KUKA KRL program: CadMatchExample.src, CadMatchExample.dat

--- CadMatchExample.src ---
&ACCESS RVO
&REL 1
&PARAM DISKPATH = KRC:\R1\Program

DEF CadMatchExample()
   ;------------------------------------------------------------------------
   ; CADMatch Example Program for Roboception rc_visard/rc_cube
   ;
   ; This program demonstrates CAD-based object detection and pick-and-place
   ; operations using Roboception's CADMatch module. The program:
   ; 1. Configures detection parameters for the specified template
   ; 2. Performs object detection with retry mechanism
   ; 3. Executes pick-and-place operations for detected objects
   ; 4. Continues until no more objects are found or program is interrupted
   ;
   ; IMPORTANT SETUP INSTRUCTIONS:
   ; 1. The service names MUST match exactly with your EKI XML configuration files
   ; 2. Modify only the parameters in this section before running the program
   ; 3. Teach the STARTPOSE and PLACEPOSE positions in the .dat file
   ; 4. Define the GripperClose() and GripperOpen() functions for your specific gripper
   ;
   ; HOW THE PROGRAM WORKS:
   ; - The program calls the CADMatch detection service which returns an array of possible grasps
   ; - Currently, only the first grasp (index 1) is used for the pick-and-place sequence
   ; - The program reads the gripper_id associated with the first grasp.
   ; - Based on the gripper_id, a target opening value is determined.
   ; - If detection fails, the program will retry up to MAX_DETECTION_RETRIES times
   ; - After successful detection, the robot will:
   ;   a) Move to a pre-grasp position above the detected object
   ;   b) Move down to grasp the object
   ;   c) Pick up the object and move to the pre-place position
   ;   d) Place the object at the taught PLACEPOSE
   ;   e) Return to the start position and repeat the cycle
   ;
   ; To use multiple detected objects, you would need to modify the code to
   ; iterate through the DETECTEDGRASPS array (indices 1 to NUMDETECTEDGRASPS)
   ;------------------------------------------------------------------------
   DECL INT MAX_DETECTION_RETRIES
   DECL INT RETRY_COUNT
   DECL REAL targetOpening      ; Calculated target opening for the gripper
   DECL REAL defaultOpening     ; Default opening value
   DECL CHAR tempMsg[120]       ; Temporary buffer for constructing messages
   DECL STATE_T State           ; State variable for SWRITE
   DECL INT Offset              ; Offset variable for SWRITE
   DECL E6POS selectedPlacePose ; Stores the selected place pose

   ; Service name - same as the EKI service name
   ; TODO: Change this to the correct service name - could be "sensor_a_pipeline_1_rc_cadmatch-detect_object"
   serviceNameDetect[] = "rc_cadmatch-detect_object"
   serviceNameStart[] = "rc_cadmatch-start"
   serviceNameStop[] = "rc_cadmatch-stop"

   ; Detection configuration parameters
   TEMPLATE_ID[] = "Template_Name"         ; CAD template to match
   POSE_FRAME[] = "external"               ; Reference frame for poses
   LOAD_CARRIER_ID[] = " "                 ; Load carrier ID (Whitespace " " = none)
   ROI_ID[] = " "                          ; Region of interest ID

   ; Collision checking parameters - deactivate all to disable collision checking
   GRIPPER_ID[] = " "                      ; Gripper ID for collision checking
   ; Pre-grasp offset for collision checking (in meters) - negtive vlaues normally desired
   PRE_GRASP_OFFSET_X = 0.0                 ; X offset - set to 0 to disable
   PRE_GRASP_OFFSET_Y = 0.0                 ; Y offset - set to 0 to disable
   PRE_GRASP_OFFSET_Z = -0.3                ; Z offset - set to 0 to disable

   ; Motion parameters (in millimeters)
   MOT_PRE_GRASP_Z_OFFSET = -300        ; Vertical offset for pre-grasp position
   MOT_PRE_PLACE_Z_OFFSET = -300        ; Vertical offset for pre-place position

   ; Detection retry configuration
   MAX_DETECTION_RETRIES = 3        ; Maximum number of detection attempts

   ; Gripper configuration
   defaultOpening = 100.0           ; Set your default gripper opening here

   ; Initialize robot and set up interrupts
   ;FOLD INI
      ;FOLD BASISTECH INI
         GLOBAL INTERRUPT DECL 3 WHEN $STOPMESS==TRUE DO IR_STOPM()
         INTERRUPT ON 3
         BAS(#INITMOV,0)
      ;ENDFOLD (BASISTECH INI)
   ;ENDFOLD (INI)

   ; Initialize message received interrupt for EKI communication
   INTERRUPT DECL 89 WHEN $FLAG[998] DO RC_NOTIFYRECEIVED(1, 998)
   INTERRUPT ON 89

   ; Move robot to home position and open gripper
   GripperOpen(defaultOpening)
   MoveToStartPosition()

   ; Initialize CADMatch module and open connection to rc_cube
   RC_START(serviceNameStart[])
   $FLAG[1] = FALSE
   RC_SETMSG("Start")

   RC_INIT(serviceNameDetect[])

   ; Main detection and pick-and-place loop
   LOOP
      ; Reset vision results
      ResetDetectedGrasps()
      RECEIVED_GRIPPER_ID[] = "none" ; Reset received ID for this cycle
      RECEIVED_GRASP_ID[] = "none"   ; Reset received grasp ID for this cycle
      targetOpening = defaultOpening   ; Reset target opening to default

      ; Attempt detection with retries
      FOR RETRY_COUNT = 1 TO MAX_DETECTION_RETRIES
         ; Pass all parameters to PerformDetection
         PerformDetection(serviceNameDetect[], TEMPLATE_ID[], POSE_FRAME[], LOAD_CARRIER_ID[], ROI_ID[], GRIPPER_ID[], PRE_GRASP_OFFSET_X, PRE_GRASP_OFFSET_Y, PRE_GRASP_OFFSET_Z)

         IF DetectionSuccessful() THEN
            RC_SETMSG("Detection successful")
            EXIT
         ENDIF

         IF RETRY_COUNT < MAX_DETECTION_RETRIES THEN
            ; Display the specific error message from RETURNCODE instead of generic one
            Offset = 0 ; Reset SWRITE offset
            SWRITE(tempMsg[], State, Offset, "Detection failed (Attempt %d/%d): %s Retrying...", RETRY_COUNT, MAX_DETECTION_RETRIES, RETURNCODE.MSG[])
            RC_SETMSG(tempMsg[])
            WAIT SEC 1.0  ; Brief delay between retries
         ENDIF
      ENDFOR

      IF DetectionSuccessful() THEN
         ; --- Gripper ID Logic ---
         ; Print the received gripper ID
         Offset = 0 ; Reset offset for SWRITE
         SWRITE(tempMsg[], State, Offset, "Received Gripper ID: %s", RECEIVED_GRIPPER_ID[])
         RC_SETMSG(tempMsg[])

         ; Print the received grasp ID
         Offset = 0 ; Reset offset for SWRITE
         SWRITE(tempMsg[], State, Offset, "Received Grasp ID: %s", RECEIVED_GRASP_ID[])
         RC_SETMSG(tempMsg[])

         ; Determine target opening based on ID
         IF STRCOMP(RECEIVED_GRIPPER_ID[], "gripper_a", #NOT_CASE_SENS) THEN
            targetOpening = 100.0
            RC_SETMSG("Gripper A identified, setting opening to 100.0")
         ELSE
            IF STRCOMP(RECEIVED_GRIPPER_ID[], "gripper_b", #NOT_CASE_SENS) THEN
               targetOpening = 50.0
               RC_SETMSG("Gripper B identified, setting opening to 50.0")
            ELSE
               ; Handle unknown or default case ("none" or other IDs)
               targetOpening = defaultOpening ; Use default opening
               RC_SETMSG("Unknown or default gripper ID, using default opening.")
            ENDIF
         ENDIF
         ; --- End Gripper ID Logic ---

         ; --- Place Pose Selection Logic based on Grasp ID ---

         IF STRCOMP(RECEIVED_GRASP_ID[], "grasp_1", #NOT_CASE_SENS) THEN
            selectedPlacePose = PLACEPOSE1 ; Assumes PLACEPOSE1 is defined in .dat
            RC_SETMSG("Grasp ID grasp_1 detected, using PLACEPOSE1.")
         ELSE
            IF STRCOMP(RECEIVED_GRASP_ID[], "grasp_2", #NOT_CASE_SENS) THEN
               selectedPlacePose = PLACEPOSE2 ; Assumes PLACEPOSE2 is defined in .dat
               RC_SETMSG("Grasp ID grasp_2 detected, using PLACEPOSE2.")
            ELSE
               selectedPlacePose = PLACEPOSE ; Use original PLACEPOSE as default
               RC_SETMSG("Unknown or default grasp ID, using default PLACEPOSE.")
            ENDIF
         ENDIF
         ; --- End Place Pose Selection Logic ---

         ExecutePickAndPlace(DETECTEDGRASPS[1], selectedPlacePose, MOT_PRE_GRASP_Z_OFFSET, MOT_PRE_PLACE_Z_OFFSET, targetOpening)
      ELSE
         HandleDetectionFailure()
         EXIT  ; Exit main loop if detection fails after all retries
      ENDIF
   ENDLOOP

   ; Clean up and stop the service
   RC_STOP(serviceNameStop[])
END

DEF ExecutePickAndPlace(GRASPPOSE:IN, PLACEPOSE:IN, MOT_PRE_GRASP_Z_OFFSET:IN, MOT_PRE_PLACE_Z_OFFSET:IN, targetOpening:IN)
   ; Executes a complete pick-and-place operation
   ;
   ; @param GRASPPOSE: Target pose for grasping the object
   ; @param PLACEPOSE: Target pose for placing the object
   ; @param MOT_PRE_GRASP_Z_OFFSET: Vertical offset (mm) for pre-grasp approach position
   ; @param MOT_PRE_PLACE_Z_OFFSET: Vertical offset (mm) for pre-place approach position
   ; @param targetOpening: The calculated opening value for the gripper

   DECL FRAME GRASPPOSE
   DECL E6POS PLACEPOSE
   DECL REAL MOT_PRE_GRASP_Z_OFFSET, MOT_PRE_PLACE_Z_OFFSET
   DECL REAL targetOpening

   ; Internal pose calculations
   DECL FRAME PREGRASPPOSE, PREPLACEPOSE
   DECL FRAME F_OFFSET

   ; Calculate pre-grasp pose using frame offset
   F_OFFSET = $NULLFRAME
   F_OFFSET.Z = MOT_PRE_GRASP_Z_OFFSET
   PREGRASPPOSE = GRASPPOSE:F_OFFSET

   ; Calculate pre-place pose
   PREPLACEPOSE = PLACEPOSE
   PREPLACEPOSE.z = PLACEPOSE.z + MOT_PRE_PLACE_Z_OFFSET

   ; Move to pre-grasp position
   SPTP PREGRASPPOSE WITH $VEL_AXIS[1] = SVEL_JOINT(rptpVelocityStd), $TOOL = STOOL2(fDatDefault), $BASE = SBASE(fDatDefault.BASE_NO), $IPO_MODE = SIPO_MODE(fDatDefault.IPO_FRAME), $LOAD = SLOAD(fDatDefault.TOOL_NO), $ACC_AXIS[1] = SACC_JOINT(pDatDefault), $APO = SAPO_PTP(pDatDefault), $GEAR_JERK[1] = SGEAR_JERK(pDatDefault)

   ; Open gripper before final approach (optional, might be already open)
   ; GripperOpen(targetOpening) ; Consider if needed here or rely on initial open

   ; Move to grasp position
   SLIN GRASPPOSE WITH $VEL = SVEL_CP(rlinVelocitySlow, , lDatDefault), $TOOL = STOOL2(fDatDefault), $BASE = SBASE(fDatDefault.BASE_NO)

   ; Activate gripper
   GripperClose()

   ; Add a small wait if needed for gripper to physically close
   WAIT SEC 0.5 ; Adjust timing as needed

   ; Optional: Add grasp check logic here if available for your gripper

   ; Move back to pre-grasp position
   SLIN PREGRASPPOSE WITH $VEL = SVEL_CP(rlinVelocityStd, , lDatDefault), $TOOL = STOOL2(fDatDefault), $BASE = SBASE(fDatDefault.BASE_NO)

   ; Move to pre-place position
   SPTP PREPLACEPOSE WITH $VEL_AXIS[1] = SVEL_JOINT(rptpVelocityStd), $TOOL = STOOL2(fDatDefault), $BASE = SBASE(fDatDefault.BASE_NO), $IPO_MODE = SIPO_MODE(fDatDefault.IPO_FRAME), $LOAD = SLOAD(fDatDefault.TOOL_NO), $ACC_AXIS[1] = SACC_JOINT(pDatDefault), $APO = SAPO_PTP(pDatDefault), $GEAR_JERK[1] = SGEAR_JERK(pDatDefault)

   ; Move to place position (user-taught position)
   ;FOLD LIN PLACEPOSE Vel=0.2 m/s CPDAT1 Tool[0]:Magnet Base[0] ;%{PE}
      ;FOLD Parameters ;%{h}
         ;Params IlfProvider=kukaroboter.basistech.inlineforms.movement.old; Kuka.IsGlobalPoint=False; Kuka.PointName=P4; Kuka.BlendingEnabled=False; Kuka.MoveDataName=CPDAT1; Kuka.VelocityPath=0.2; Kuka.CurrentCDSetIndex=0; Kuka.MovementParameterFieldEnabled=True; IlfCommand=LIN
      ;ENDFOLD
      $BWDSTART = FALSE
      LDAT_ACT = lDatDefault
      FDAT_ACT = fDatDefault
      BAS(#CP_PARAMS, 0.2)
      SET_CD_PARAMS(0)
      LIN PLACEPOSE
   ;ENDFOLD

   ; Release object
   GripperOpen(targetOpening)

   ; Add a small wait if needed for gripper to physically open
   WAIT SEC 0.5 ; Adjust timing as needed

   ; Move back to pre-place position
   SLIN PREPLACEPOSE WITH $VEL = SVEL_CP(rlinVelocityStd, , lDatDefault), $TOOL = STOOL2(fDatDefault), $BASE = SBASE(fDatDefault.BASE_NO)

   ; Return to home position
   MoveToStartPosition()
END

; ---- Helper Functions ----
DEF MoveToStartPosition()
   ;FOLD SPTP STARTPOSE Vel=100 % DEFAULT
      SPTP STARTPOSE WITH $VEL_AXIS[1]= SVEL_JOINT(100), $TOOL= STOOL2(fDatDefault), $BASE= SBASE(fDatDefault.BASE_NO), $IPO_MODE= SIPO_MODE(fDatDefault.IPO_FRAME), $LOAD= SLOAD(fDatDefault.TOOL_NO), $ACC_AXIS[1]= SACC_JOINT(PDEFAULT), $GEAR_JERK[1]= SGEAR_JERK(PDEFAULT)
   ;ENDFOLD
END

DEF GripperClose()
   ; Implement gripper closing logic here
   RC_SETMSG("Gripper closing")
   ; Example: SetOutput(GripperCloseSignal, TRUE)
   ; Example: SetOutput(GripperOpenSignal, FALSE)
   WAIT SEC 0.1 ; Add delay if needed
END

DEF GripperOpen(targetOpening:IN)
   ; Implement gripper opening logic here, using the targetOpening value
   DECL REAL targetOpening
   DECL KrlMsgPar_T params[1]

   ; Setup parameter for message
   params[1] = {par_type #VALUE, par_real 0}
   params[1].par_real = targetOpening

   RC_SETMSG_PARAM("Gripper opening to %1", params[])
   ; Example: SetAnalogOutput(GripperPositionSignal, targetOpening)
   ; Example: SetOutput(GripperCloseSignal, FALSE)
   ; Example: SetOutput(GripperOpenSignal, TRUE)
   WAIT SEC 0.1 ; Add delay if needed
END

; ---- Roboception Functions ----
;FOLD ROBOCEPTION_FUNCTIONS
   DEF PerformDetection(serviceNameDetect[]:IN, TEMPLATE_ID[]:IN, POSE_FRAME[]:IN, LOAD_CARRIER_ID[]:IN, ROI_ID[]:IN, GRIPPER_ID[]:IN, PRE_GRASP_OFFSET_X:IN, PRE_GRASP_OFFSET_Y:IN, PRE_GRASP_OFFSET_Z:IN)
      DECL CHAR serviceNameDetect[]
      DECL EKI_STATUS RET
      DECL CHAR TEMPLATE_ID[]
      DECL CHAR POSE_FRAME[]
      DECL CHAR LOAD_CARRIER_ID[]
      DECL CHAR ROI_ID[]
      DECL CHAR GRIPPER_ID[]
      DECL REAL PRE_GRASP_OFFSET_X
      DECL REAL PRE_GRASP_OFFSET_Y
      DECL REAL PRE_GRASP_OFFSET_Z
      DECL E6POS flangePose

      flangePose = $POS_ACT_MES : INV_POS($TOOL)

      RET = EKI_SetString(serviceNameDetect[], "req/args/template_id", TEMPLATE_ID[])
      RET = EKI_SetString(serviceNameDetect[], "req/args/pose_frame", POSE_FRAME[])
      RET = EKI_SetFrame(serviceNameDetect[], "req/args/robot_pose", flangePose)

      IF LOAD_CARRIER_ID[1] <> " " THEN
         RET = EKI_SetString(serviceNameDetect[], "req/args/load_carrier_id", LOAD_CARRIER_ID[])
      ENDIF

      IF ROI_ID[1] <> " " THEN
         RET = EKI_SetString(serviceNameDetect[], "req/args/region_of_interest_id", ROI_ID[])
      ENDIF

      IF GRIPPER_ID[1] <> " " THEN
         RET = EKI_SetString(serviceNameDetect[], "req/args/collision_detection/@gripper_id", GRIPPER_ID[])
      ENDIF

      IF PRE_GRASP_OFFSET_X <> 0.0 THEN
         RET = EKI_SetReal(serviceNameDetect[], "req/args/collision_detection/pre_grasp_offset/@x", PRE_GRASP_OFFSET_X)
      ENDIF

      IF PRE_GRASP_OFFSET_Y <> 0.0 THEN
         RET = EKI_SetReal(serviceNameDetect[], "req/args/collision_detection/pre_grasp_offset/@y", PRE_GRASP_OFFSET_Y)
      ENDIF

      IF PRE_GRASP_OFFSET_Z <> 0.0 THEN
         RET = EKI_SetReal(serviceNameDetect[], "req/args/collision_detection/pre_grasp_offset/@z", PRE_GRASP_OFFSET_Z)
      ENDIF

      ; Open connection before sending request
      RC_OPENCONNECTION(serviceNameDetect[])

      ; Force synchronization
      WAIT SEC 0

      ; Send request
      RET = EKI_Send(serviceNameDetect[], "req")

      ; Wait for response
      RC_WAITFORRESULT(1)

      ; Read results
      RC_READRESULT(serviceNameDetect[])

      ; Close the connection after reading results
      RC_CLOSECONNECTION(serviceNameDetect[], "req")
   END

   DEFFCT BOOL DetectionSuccessful()
      DECL KrlMsgPar_T params[1]

      IF (RETURNCODE.VALUE < 0) THEN
         RETURN FALSE
      ENDIF

      IF CheckDetectedItem(1) THEN
         ; Show number of detected grasps
         params[1] = {par_type #VALUE, par_real 0}
         params[1].par_real = NUMDETECTEDGRASPS
         RC_SETMSG_PARAM("%1 grasps detected", params[])
         RETURN TRUE
      ENDIF

      RETURN FALSE
   ENDFCT

   DEFFCT BOOL CheckDetectedItem(Index:IN)
      DECL INT Index
      DECL KrlMsgPar_T par[3]

      IF (DETECTEDGRASPS[Index].X == 0) AND (DETECTEDGRASPS[Index].Y == 0) AND (DETECTEDGRASPS[Index].Z == 0) AND (DETECTEDGRASPS[Index].A == 0) AND (DETECTEDGRASPS[Index].B == 0) AND (DETECTEDGRASPS[Index].C ==0) THEN
         RETURN FALSE
      ELSE
         ;Show cad match pose
         par[1] = {par_type #value, par_real 0}
         par[1].par_real = DETECTEDGRASPS[1].X
         par[2] = {par_type #value, par_real 0}
         par[2].par_real = DETECTEDGRASPS[1].Y
         par[3] = {par_type #value, par_real 0}
         par[3].par_real = DETECTEDGRASPS[1].Z
         RC_SETMSG_PARAM("Grasp pose: X: %1, Y: %2, Z: %3", par[])
         RETURN TRUE
      ENDIF
   ENDFCT

   DEF HandleDetectionFailure()
      IF (RETURNCODE.VALUE > 0) THEN
         RC_SETMSG("No CADMatch result")
      ENDIF
      HALT
   END

   DEF RC_SETMSG(msg[]:IN)
      DECL CHAR msg[]
      DECL KrlMsgPar_T params[3]

      RC_SETMSG_PARAM(msg[], params[])
   END

   DEF RC_SETMSG_PARAM(msg[]:IN, params:OUT)
      DECL CHAR msg[]
      DECL KrlMsgPar_T params[]

      DECL KrlMsg_T name
      DECL KrlMsgOpt_T options
      DECL INT Handle, len, count
      DECL EKrlMsgType Type

      name={modul[] "rc", nr 1, msg_txt[] " "}

      Type=#notify

      len=STRLEN(msg[])
      IF len>0 THEN
         IF len>80 THEN
            len=80
         ENDIF
         FOR count=1 TO len
            name.msg_txt[count]=msg[count]
         ENDFOR
      ELSE
         name.msg_txt[]="parameter msg[] is missing"
      ENDIF

      Handle=Set_KrlMsg(Type, name, params[], options)
   END

   DEF RC_INIT(configFileName[]:IN)
      DECL CHAR configFileName[]
      DECL EKI_Status RET

      RET=EKI_INIT(configFileName[])
   END

   DEF RC_OPENCONNECTION(configFileName[]:IN)
      DECL CHAR configFileName[]
      DECL EKI_Status RET

      RET=EKI_Open(configFileName[])
      EKI_CHECK(RET,#Quit)
   END

   DEF RC_CLOSECONNECTION(configFileName[]:IN, strPlace[]:IN)
      DECL CHAR configFileName[]
      DECL CHAR strPlace[]
      DECL EKI_Status RET

      WAIT SEC 0
      RET=EKI_Close(configFileName[])
      RET=EKI_ClearBuffer(configFileName[], strPlace[])
   END

   DEF RC_WAITFORRESULT(WaitFlag:IN)
      DECL INT WaitFlag

      WAIT FOR $FLAG[WaitFlag] OR NOT $FLAG[RCEkiAliveFlagNo]
      ;Eki-connection has been closed
      IF(NOT $FLAG[RCEkiAliveFlagNo]) THEN
         RC_SETMSG("EKI connection lost")
      ENDIF

      $FLAG[WaitFlag] = FALSE
      WAIT SEC 0
   END

   DEF RC_NOTIFYRECEIVED(WAITFLAG:IN, EOFRESULFLAG:IN)
      DECL INT WAITFLAG
      DECL INT EOFRESULFLAG

      $FLAG[EOFRESULFLAG]=FALSE
      $FLAG[WAITFLAG]=TRUE
   END

   DEF RC_READRESULT(configFileName[]:IN)
      DECL CHAR configFileName[]
      DECL RETURNCODE_T RESULT
      DECL EKI_STATUS RET
      DECL INT j
      DECL FRAME POSE

      POSE = POSE_IDENT
      RESULT={VALUE 0, MSG[] "0"}
      RECEIVED_GRIPPER_ID[] = "none"
      RECEIVED_GRASP_ID[] = "none" ; Initialize grasp ID

      ;Receive error codes
      RET = EKI_GetInt(configFileName[], "res/return_code/@value", RESULT.VALUE)
      RET = EKI_GetString(configFileName[], "res/return_code/@message", RESULT.MSG[])
      RETURNCODE = RESULT

      ; Display error message immediately if there is one
      IF (RESULT.VALUE < 0) THEN
         RC_SETMSG("API Error")
         RC_SETMSG(RESULT.MSG[])
      ENDIF

      ;Receive number of detections
      RET = EKI_CheckBuffer(configFileName[], "res/grasps/le/id")
      NUMDETECTEDGRASPS = RET.Buff

      ;Receive frames
      FOR j=1 to NUMDETECTEDGRASPS
         RET = EKI_GetFrame(configFileName[], "res/grasps/le/pose", POSE)
         DETECTEDGRASPS[j] = POSE
         ; For the first grasp (j=1), also read its gripper_id and grasp_id
         IF j == 1 THEN
            ; Read the gripper_id associated with the first grasp
            RET = EKI_GetString(configFileName[], "res/grasps/le/gripper_id", RECEIVED_GRIPPER_ID[])
            ; Read the id (grasp_id) associated with the first grasp
            RET = EKI_GetString(configFileName[], "res/grasps/le/id", RECEIVED_GRASP_ID[])
         ENDIF
      ENDFOR
      RET = EKI_ClearBuffer(configFileName[], "res")
   END

   DEF RC_START(serviceNameStart[]:IN)
      DECL CHAR serviceNameStart[]
      DECL EKI_Status RET

      $FLAG[1] = FALSE
      RC_SETMSG("Start")
      RC_INIT(serviceNameStart[])
      RC_OPENCONNECTION(serviceNameStart[])
      RET = EKI_Send(serviceNameStart[], "req")
      RC_WAITFORRESULT(1)
      RC_CLOSECONNECTION(serviceNameStart[], "req")
   END

   DEF RC_STOP(serviceNameStop[]:IN)
      DECL CHAR serviceNameStop[]
      DECL EKI_Status RET

      $FLAG[1] = FALSE
      RC_SETMSG("Stop")
      RC_INIT(serviceNameStop[])
      RC_OPENCONNECTION(serviceNameStop[])
      RET = EKI_Send(serviceNameStop[], "req")
      RC_WAITFORRESULT(1)
      RC_CLOSECONNECTION(serviceNameStop[], "req")
   END

   DEF ResetDetectedGrasps()
      DECL INT I

      FOR I = 1 TO 32 STEP 1
         DETECTEDGRASPS[I]=$NULLFRAME
      ENDFOR
   END
;ENDFOLD (ROBOCEPTION_FUNCTIONS)

--- CadMatchExample.dat ---
&ACCESS RVO
&REL 1
&PARAM DISKPATH = KRC:\R1\Program

DEFDAT  CADMATCHEXAMPLE

   ;FOLD EXTERNAL DECLARATIONS;%{PE}%MKUKATPBASIS,%CEXT,%VCOMMON,%P
   ;FOLD BASISTECH EXT;%{PE}%MKUKATPBASIS,%CEXT,%VEXT,%P
   EXT  BAS (BAS_COMMAND  :IN,REAL  :IN )
   ;ENDFOLD (BASISTECH EXT)
   ;FOLD USER EXT;%{E}%MKUKATPUSER,%CEXT,%VEXT,%P
   ;Make your modifications here

   ; Common structures and variables
   STRUC RETURNCODE_T INT VALUE,CHAR MSG[512]
   DECL INT RCEkiAliveFlagNo=997
   DECL RETURNCODE_T RETURNCODE
   DECL FRAME POSE_IDENT={X 0.0,Y 0.0,Z 0.0,A 0.0,B 0.0,C 0.0}

   ; Service configuration
   DECL CHAR serviceNameDetect[64]
   DECL CHAR serviceNameStart[64]
   DECL CHAR serviceNameStop[64]

   ; Detection parameters
   DECL CHAR TEMPLATE_ID[60]
   DECL CHAR POSE_FRAME[32]
   DECL CHAR LOAD_CARRIER_ID[32]
   DECL CHAR ROI_ID[32]
   DECL CHAR GRIPPER_ID[32] ; Stores the ID of the gripper
   DECL CHAR RECEIVED_GRASP_ID[32] ; Stores the ID of the received grasp
   DECL REAL PRE_GRASP_OFFSET_X
   DECL REAL PRE_GRASP_OFFSET_Y
   DECL REAL PRE_GRASP_OFFSET_Z
   DECL REAL MOT_PRE_GRASP_Z_OFFSET
   DECL REAL MOT_PRE_PLACE_Z_OFFSET

   ; Detection results
   DECL FRAME DETECTEDGRASPS[32]
   DECL CHAR RECEIVED_GRIPPER_ID[32]
   DECL INT NUMDETECTEDGRASPS

   ; Robot parameters
   DECL REAL rlinVelocityStd=0.25    ; m/s
   DECL REAL rlinVelocitySlow=0.15   ; m/s
   DECL REAL rptpVelocityStd=10      ; %

   ; Position data - teach these poses
   DECL E6POS STARTPOSE={X 0,Y 0,Z 0,A 0,B 0,C 0,S 0,T 0,E1 0.0,E2 0.0,E3 0.0,E4 0.0,E5 0.0,E6 0.0}
   DECL E6POS PLACEPOSE={X 0,Y 0,Z 0,A 0,B 0,C 0,S 0,T 0,E1 0.0,E2 0.0,E3 0.0,E4 0.0,E5 0.0,E6 0.0}
   DECL E6POS PLACEPOSE1={X 0,Y 0,Z 0,A 0,B 0,C 0,S 0,T 0,E1 0.0,E2 0.0,E3 0.0,E4 0.0,E5 0.0,E6 0.0}
   DECL E6POS PLACEPOSE2={X 0,Y 0,Z 0,A 0,B 0,C 0,S 0,T 0,E1 0.0,E2 0.0,E3 0.0,E4 0.0,E5 0.0,E6 0.0}


   ; Movement data
   DECL LDAT lDatDefault={VEL 2.00000,ACC 20.0000,APO_DIST 10.0000,APO_FAC 50.0000,AXIS_VEL 100.000,AXIS_ACC 100.000,ORI_TYP #VAR,CIRC_TYP #BASE,JERK_FAC 50.0000,GEAR_JERK 100.000,EXAX_IGN 0,CB {AUX_PT {ORI #CONSIDER,E1 #CONSIDER,E2 #CONSIDER,E3 #CONSIDER,E4 #CONSIDER,E5 #CONSIDER,E6 #CONSIDER},TARGET_PT {ORI #INTERPOLATE,E1 #INTERPOLATE,E2 #INTERPOLATE,E3 #INTERPOLATE,E4 #INTERPOLATE,E5 #INTERPOLATE,E6 #INTERPOLATE}}}
   DECL FDAT fDatDefault={TOOL_NO 4,BASE_NO 0,IPO_FRAME #BASE,POINT2[] " "}
   DECL PDAT pDatDefault={VEL 10.0000,ACC 20.0000,APO_DIST 10.0000,APO_MODE #CDIS,GEAR_JERK 100.000,EXAX_IGN 0}

   ;ENDFOLD (USER EXT)
   ;ENDFOLD (EXTERNAL DECLARATIONS)
ENDDAT
